PROGRAM Rotina019_Manual
VAR
	status: INT;
	
	posicaoAtual: STRING;
	envialog: STRING;
	
	fbTimeVentila: ton;
	fbTimeAqueci: ton;
	
	totalManual: STRING(255);
	tempo: STRING(255);
END_VAR

fbTimeVentila();
fbTimeAqueci();

CASE status OF

0:
IF gvl_p.arrStatusEstufas[0].startManual AND STRING_TO_DT(gvl.progInicio[0]) <= systemtime_to_dt(gvl.fbGetLocalSystemTime.systemTime)  THEN
	status:= 5;
	
	gvl.bstartchart019:= TRUE;
	gvl_p.zona1setpt_019:= gvl_p.arr_CustomTime[0,1];
	gvl_p.zona2setpt_019:= gvl_p.arr_CustomTime[0,1];
	gvl.liga_ventilacao_019:= TRUE;
	fbTimeVentila(in:= TRUE, pt:=T#1S);
	
///// GERADOR DE LOG -------------------------------------------------------------

envialog:= 'Programação Manual Iniciada ESTUFA 019';
gvl.logRegister19:= envialog;

	gvl_p.etapa_process[0] := 'Inicializando';
	
ELSE
	status:= 0;
	IF gvl_p.arrStatusEstufas[0].start THEN
		gvl_p.etapa_process[0] := gvl.progInicio[0];
	END_IF
END_IF
5:
IF fbTimeVentila.Q THEN
	status:= 10;
	gvl.liga_ventilacao_019:=FALSE;
	fbTimeVentila(in:= FALSE);
ELSE
	status:= 5;
END_IF

10:
IF gvl.ventilacao_Ligada_019 THEN
	status:= 15;
	
	gvl.liga_aquecimento_019:= TRUE;
	fbTimeAqueci(in:= TRUE, pt:= T#1S);
	
///// GERADOR DE LOG -------------------------------------------------------------

envialog:= 'Aquecendo ESTUFA 019';
gvl.logRegister19:= envialog;
	
	gvl_p.etapa_process[0] := 'Aquecendo';
	
ELSE
	status:= 10;
END_IF

15:
IF fbTimeAqueci.Q THEN
	status:= 20;
	
	gvl.liga_aquecimento_019:= FALSE;
	fbTimeAqueci(in:=false);
ELSE
	status:= 15;
END_IF

20:
IF gvl.zona1atual_019 >= gvl_p.zona1setpt_019 THEN
	status:= 30;
	
gvl.progInicio[0]:= DT_TO_STRING(gvl.somaTempo);
	
///// CALCULAR FIM DA SECAGEM E DA ARMAZENAGEM --------------------------------------------------------------------------------

totalManual:= insert('T#h',INT_TO_STRING(gvl.totalManual[0]),2);
gvl_p.arrStatusEstufas[0].inicioSecagem := STRING_TO_DT(gvl.progInicio[0]);
gvl_p.arrStatusEstufas[0].fimSecagem := STRING_TO_DT(gvl.progInicio[0]) + STRING_TO_TIME(totalManual);
gvl_P.arrStatusEstufas[0].prevFimSeca := gvl_p.arrStatusEstufas[0].fimSecagem;
//gvl_p.arrStatusEstufas[0].fimArmazenagem := gvl_p.arrStatusEstufas[0].fimSecagem + gvl_p.arrStatusEstufas[0].tempoArmazenagem ;

///// IMPRIMIR A HORA E A DATA DO INICIO DA SECAGEM ---------------------------------------------------------------------------
gvl_p.arrStatusEstufas[0].statusInicioSecagem := '';
gvl_p.arrStatusEstufas[0].statusInicioSecagem := concat(gvl_p.arrStatusEstufas[0].statusInicioSecagem,gvl.hora);
gvl_p.arrStatusEstufas[0].statusInicioSecagem := concat(gvl_p.arrStatusEstufas[0].statusInicioSecagem,':');
gvl_p.arrStatusEstufas[0].statusInicioSecagem := concat(gvl_p.arrStatusEstufas[0].statusInicioSecagem,gvl.minuto);
gvl_p.arrStatusEstufas[0].statusInicioSecagem := concat(gvl_p.arrStatusEstufas[0].statusInicioSecagem,' ');
gvl_p.arrStatusEstufas[0].statusInicioSecagem := concat(gvl_p.arrStatusEstufas[0].statusInicioSecagem,gvl.dia);
gvl_p.arrStatusEstufas[0].statusInicioSecagem := concat(gvl_p.arrStatusEstufas[0].statusInicioSecagem,'/');
gvl_p.arrStatusEstufas[0].statusInicioSecagem := concat(gvl_p.arrStatusEstufas[0].statusInicioSecagem,gvl.mes);
gvl_p.arrStatusEstufas[0].statusInicioSecagem := concat(gvl_p.arrStatusEstufas[0].statusInicioSecagem,'/');
gvl_p.arrStatusEstufas[0].statusInicioSecagem := concat(gvl_p.arrStatusEstufas[0].statusInicioSecagem,gvl.ano);

//--------------------REATOR------------------------------------

IF gravarConfigPosicao_Reator.bGravarConfigPosicao_Reator THEN
	gvl_p.arrStatusEstufas[0].inicioReator := '';
	gvl_p.arrStatusEstufas[0].inicioReator := concat(gvl_p.arrStatusEstufas[0].inicioReator,gvl.hora);
	gvl_p.arrStatusEstufas[0].inicioReator := concat(gvl_p.arrStatusEstufas[0].inicioReator,':');
	gvl_p.arrStatusEstufas[0].inicioReator := concat(gvl_p.arrStatusEstufas[0].inicioReator,gvl.minuto);
	gvl_p.arrStatusEstufas[0].inicioReator := concat(gvl_p.arrStatusEstufas[0].inicioReator,' ');
	gvl_p.arrStatusEstufas[0].inicioReator := concat(gvl_p.arrStatusEstufas[0].inicioReator,gvl.dia);
	gvl_p.arrStatusEstufas[0].inicioReator := concat(gvl_p.arrStatusEstufas[0].inicioReator,'/');
	gvl_p.arrStatusEstufas[0].inicioReator := concat(gvl_p.arrStatusEstufas[0].inicioReator,gvl.mes);
	gvl_p.arrStatusEstufas[0].inicioReator := concat(gvl_p.arrStatusEstufas[0].inicioReator,'/');
	gvl_P.arrStatusEstufas[0].inicioReator := concat(gvl_p.arrStatusEstufas[0].inicioReator,gvl.ano);
END_IF

///// DECOMPOR A VARIAVEL FIM DA SECAGEM -----------------------------------------------------------------------------------------------
gvl_p.arrStatusEstufas[0].diaSec := MID(STR:= DT_TO_STRING(gvl_p.arrStatusEstufas[0].fimSecagem) , LEN:= 2, POS:=12);
gvl_p.arrStatusEstufas[0].mesSec := MID(STR:= DT_TO_STRING(gvl_p.arrStatusEstufas[0].fimSecagem), LEN:= 2, POS:=9);
gvl_p.arrStatusEstufas[0].anoSec := MID(STR:= DT_TO_STRING(gvl_p.arrStatusEstufas[0].fimSecagem), LEN:= 2, POS:=6);
gvl_p.arrStatusEstufas[0].horaSec := MID(STR:= DT_TO_STRING(gvl_p.arrStatusEstufas[0].fimSecagem), LEN:= 2, POS:=15);
gvl_p.arrStatusEstufas[0].minutoSec := MID(STR:= DT_TO_STRING(gvl_p.arrStatusEstufas[0].fimSecagem), LEN:= 2, POS:=18);

///// IMPRIMIR A HORA E A DATA DO FIM DA SECAGEM --------------------------------------------------------------------------------------------------------
gvl_p.arrStatusEstufas[0].statusFimSecagem := '';
gvl_p.arrStatusEstufas[0].statusFimSecagem := concat(gvl_p.arrStatusEstufas[0].statusFimSecagem,gvl_p.arrStatusEstufas[0].horaSec);
gvl_p.arrStatusEstufas[0].statusFimSecagem := concat(gvl_p.arrStatusEstufas[0].statusFimSecagem,':');
gvl_p.arrStatusEstufas[0].statusFimSecagem := concat(gvl_p.arrStatusEstufas[0].statusFimSecagem,gvl_p.arrStatusEstufas[0].minutoSec);
gvl_p.arrStatusEstufas[0].statusFimSecagem := concat(gvl_p.arrStatusEstufas[0].statusFimSecagem,' ');
gvl_p.arrStatusEstufas[0].statusFimSecagem := concat(gvl_p.arrStatusEstufas[0].statusFimSecagem,gvl_p.arrStatusEstufas[0].diaSec);
gvl_p.arrStatusEstufas[0].statusFimSecagem := concat(gvl_p.arrStatusEstufas[0].statusFimSecagem,'/');
gvl_p.arrStatusEstufas[0].statusFimSecagem := concat(gvl_p.arrStatusEstufas[0].statusFimSecagem,gvl_p.arrStatusEstufas[0].mesSec);
gvl_p.arrStatusEstufas[0].statusFimSecagem := concat(gvl_p.arrStatusEstufas[0].statusFimSecagem,'/');
gvl_p.arrStatusEstufas[0].statusFimSecagem := concat(gvl_p.arrStatusEstufas[0].statusFimSecagem,gvl_p.arrStatusEstufas[0].anoSec);


///// GERADOR DE LOG -------------------------------------------------------------
envialog:= 'Inicio T1 ESTUFA 019';
gvl.logRegister19:= envialog;

gvl_p.etapa_process[0]:= 'T1';

ELSE
	IF gvl_p.arr_CustomTime[1,1] = 0 THEN
		status:= 45;
	END_IF
	status:= 20;
END_IF

30:
tempo:= insert('T#h',INT_TO_STRING(gvl_p.arr_CustomTime[1,1]),2);
IF STRING_TO_DT(gvl.progInicio[0]) + STRING_TO_TIME(tempo) = systemtime_to_dt(gvl.fbGetLocalSystemTime.systemTime) THEN
	status:= 31;
	
	gvl_p.zona1setpt_019:= gvl_p.arr_CustomTime[0,2];
	gvl_p.zona2setpt_019:= gvl_p.arr_CustomTime[0,2];
	gvl.progInicio[0]:= DT_TO_STRING(STRING_TO_DT(gvl.progInicio[0]) + STRING_TO_TIME(tempo));
	
///// GERADOR DE LOG -------------------------------------------------------------
envialog:= 'Inicio T2 ESTUFA 019';
gvl.logRegister19:= envialog;

gvl_p.etapa_process[0]:= 'T2';
	
ELSE
	status:= 30;
END_IF

31:
tempo:= insert('T#h',INT_TO_STRING(gvl_p.arr_CustomTime[1,2]),2);
IF STRING_TO_DT(gvl.progInicio[0]) + STRING_TO_TIME(tempo) = systemtime_to_dt(gvl.fbGetLocalSystemTime.systemTime) THEN
	status:= 32;
	
	gvl_p.zona1setpt_019:= gvl_p.arr_CustomTime[0,3];
	gvl_p.zona2setpt_019:= gvl_p.arr_CustomTime[0,3];
	gvl.progInicio[0]:= DT_TO_STRING(STRING_TO_DT(gvl.progInicio[0]) + STRING_TO_TIME(tempo));
	
///// GERADOR DE LOG -------------------------------------------------------------
envialog:= 'Inicio T3 ESTUFA 019';
gvl.logRegister19:= envialog;

gvl_p.etapa_process[0]:= 'T3';
	
ELSE
	IF gvl_p.arr_CustomTime[1,2] = 0 THEN
		status:= 45;
	END_IF
	status:= 31;
END_IF

32:
tempo:= insert('T#h',INT_TO_STRING(gvl_p.arr_CustomTime[1,3]),2);
IF STRING_TO_DT(gvl.progInicio[0]) + STRING_TO_TIME(tempo) = systemtime_to_dt(gvl.fbGetLocalSystemTime.systemTime) THEN
	status:= 33;
	
	gvl_p.zona1setpt_019:= gvl_p.arr_CustomTime[0,4];
	gvl_p.zona2setpt_019:= gvl_p.arr_CustomTime[0,4];
	gvl.progInicio[0]:= DT_TO_STRING(STRING_TO_DT(gvl.progInicio[0]) + STRING_TO_TIME(tempo));
	
///// GERADOR DE LOG -------------------------------------------------------------
envialog:= 'Inicio T4 ESTUFA 019';
gvl.logRegister19:= envialog;

gvl_p.etapa_process[0]:= 'T4';
	
ELSE
	IF gvl_p.arr_CustomTime[1,3] = 0 THEN
		status:= 45;
	END_IF
	status:= 32;
END_IF

33:
tempo:= insert('T#h',INT_TO_STRING(gvl_p.arr_CustomTime[1,4]),2);
IF STRING_TO_DT(gvl.progInicio[0]) + STRING_TO_TIME(tempo) = systemtime_to_dt(gvl.fbGetLocalSystemTime.systemTime) THEN
	status:= 34;
	
	gvl_p.zona1setpt_019:= gvl_p.arr_CustomTime[0,5];
	gvl_p.zona2setpt_019:= gvl_p.arr_CustomTime[0,5];
	gvl.progInicio[0]:= DT_TO_STRING(STRING_TO_DT(gvl.progInicio[0]) + STRING_TO_TIME(tempo));
	
///// GERADOR DE LOG -------------------------------------------------------------
envialog:= 'Inicio T5 ESTUFA 019';
gvl.logRegister19:= envialog;

gvl_p.etapa_process[0]:= 'T5';
	
ELSE
	IF gvl_p.arr_CustomTime[1,4] = 0 THEN
		status:= 45;
	END_IF
	status:= 33;
END_IF

34:
tempo:= insert('T#h',INT_TO_STRING(gvl_p.arr_CustomTime[1,5]),2);
IF STRING_TO_DT(gvl.progInicio[0]) + STRING_TO_TIME(tempo) = systemtime_to_dt(gvl.fbGetLocalSystemTime.systemTime) THEN
	status:= 35;
	
	gvl_p.zona1setpt_019:= gvl_p.arr_CustomTime[0,6];
	gvl_p.zona2setpt_019:= gvl_p.arr_CustomTime[0,6];
	gvl.progInicio[0]:= DT_TO_STRING(STRING_TO_DT(gvl.progInicio[0]) + STRING_TO_TIME(tempo));
	
///// GERADOR DE LOG -------------------------------------------------------------
envialog:= 'Inicio T6 ESTUFA 019';
gvl.logRegister19:= envialog;

gvl_p.etapa_process[0]:= 'T6';
	
ELSE
	IF gvl_p.arr_CustomTime[1,5] = 0 THEN
		status:= 45;
	END_IF
	status:= 34;
END_IF

35:
tempo:= insert('T#h',INT_TO_STRING(gvl_p.arr_CustomTime[1,6]),2);
IF STRING_TO_DT(gvl.progInicio[0]) + STRING_TO_TIME(tempo) = systemtime_to_dt(gvl.fbGetLocalSystemTime.systemTime) THEN
	status:= 36;
	
	gvl_p.zona1setpt_019:= gvl_p.arr_CustomTime[0,7];
	gvl_p.zona2setpt_019:= gvl_p.arr_CustomTime[0,7];
	gvl.progInicio[0]:= DT_TO_STRING(STRING_TO_DT(gvl.progInicio[0]) + STRING_TO_TIME(tempo));
	
///// GERADOR DE LOG -------------------------------------------------------------
envialog:= 'Inicio T7 ESTUFA 019';
gvl.logRegister19:= envialog;

gvl_p.etapa_process[0]:= 'T7';
	
ELSE
	IF gvl_p.arr_CustomTime[1,6] = 0 THEN
		status:= 45;
	END_IF
	status:= 35;
END_IF

36:
tempo:= insert('T#h',INT_TO_STRING(gvl_p.arr_CustomTime[1,7]),2);
IF STRING_TO_DT(gvl.progInicio[0]) + STRING_TO_TIME(tempo) = systemtime_to_dt(gvl.fbGetLocalSystemTime.systemTime) THEN
	status:= 37;
	
	gvl_p.zona1setpt_019:= gvl_p.arr_CustomTime[0,8];
	gvl_p.zona2setpt_019:= gvl_p.arr_CustomTime[0,8];
	gvl.progInicio[0]:= DT_TO_STRING(STRING_TO_DT(gvl.progInicio[0]) + STRING_TO_TIME(tempo));
	
///// GERADOR DE LOG -------------------------------------------------------------
envialog:= 'Inicio T8 ESTUFA 019';
gvl.logRegister19:= envialog;

gvl_p.etapa_process[0]:= 'T8';
	
ELSE
	IF gvl_p.arr_CustomTime[1,7] = 0 THEN
		status:= 45;
	END_IF
	status:= 36;
END_IF

37:
tempo:= insert('T#h',INT_TO_STRING(gvl_p.arr_CustomTime[1,8]),2);
IF STRING_TO_DT(gvl.progInicio[0]) + STRING_TO_TIME(tempo) = systemtime_to_dt(gvl.fbGetLocalSystemTime.systemTime) THEN
	status:= 38;
	
	gvl_p.zona1setpt_019:= gvl_p.arr_CustomTime[0,9];
	gvl_p.zona2setpt_019:= gvl_p.arr_CustomTime[0,9];
	gvl.progInicio[0]:= DT_TO_STRING(STRING_TO_DT(gvl.progInicio[0]) + STRING_TO_TIME(tempo));
	
///// GERADOR DE LOG -------------------------------------------------------------
envialog:= 'Inicio T9 ESTUFA 019';
gvl.logRegister19:= envialog;

gvl_p.etapa_process[0]:= 'T9';
	
ELSE
	IF gvl_p.arr_CustomTime[1,8] = 0 THEN
		status:= 45;
	END_IF
	status:= 37;
END_IF

38:
tempo:= insert('T#h',INT_TO_STRING(gvl_p.arr_CustomTime[1,9]),2);
IF STRING_TO_DT(gvl.progInicio[0]) + STRING_TO_TIME(tempo) = systemtime_to_dt(gvl.fbGetLocalSystemTime.systemTime) THEN
	status:= 40;
	
	gvl_p.zona1setpt_019:= gvl_p.arr_CustomTime[0,10];
	gvl_p.zona2setpt_019:= gvl_p.arr_CustomTime[0,10];
	gvl.progInicio[0]:= DT_TO_STRING(STRING_TO_DT(gvl.progInicio[0]) + STRING_TO_TIME(tempo));
	
///// GERADOR DE LOG -------------------------------------------------------------
envialog:= 'Inicio T10 ESTUFA 019';
gvl.logRegister19:= envialog;

gvl_p.etapa_process[0]:= 'T10';
	
ELSE
	IF gvl_p.arr_CustomTime[1,9] = 0 THEN
		status:= 45;
	END_IF
	status:= 38;
END_IF

40:
tempo:= insert('T#h',INT_TO_STRING(gvl_p.arr_CustomTime[1,10]),2);
IF STRING_TO_DT(gvl.progInicio[0]) + STRING_TO_TIME(tempo) = systemtime_to_dt(gvl.fbGetLocalSystemTime.systemTime) THEN
	status:= 50;
	
	gvl_p.arrStatusEstufas[0].startManual:= FALSE;
	gvl.bstartchart019:= FALSE;
	gvl.desl_aquecimento_019:= TRUE;
	fbTimeAqueci(in:=TRUE, pt:=T#1S);
	
	gvl_p.etapa_process[0] := '';
	
	gvl_p.arrStatusEstufas[0].statusInicioSecagem := '';
	gvl_p.arrStatusEstufas[0].inicioReator := '';
	gvl_p.arrStatusEstufas[0].statusFimSecagem := '';
	gvl_p.arrStatusEstufas[0].statusFimArmazenagem := '';
	gvl_p.arrStatusEstufas[0].fimSecagem:= DT#1970-1-1-0:0:0;
	gvl.endArm19:= T#0S;
	gvl.endSeca19:= T#0S;
	
///// GERADOR DE LOG -------------------------------------------------------------
envialog:= 'Programação Finalizada ESTUFA 019';
gvl.logRegister19:= envialog;

gvl_p.etapa_process[0]:= '';

ELSE
	IF gvl_p.arr_CustomTime[1,10] = 0 THEN
		status:= 45;
	END_IF
	status:= 40;
END_IF

45:
IF gvl_p.arrStatusEstufas[0].startManual THEN
status:= 50;
	
	gvl_p.arrStatusEstufas[0].startManual:= FALSE;
	gvl.bstartchart019:= FALSE;
	gvl.desl_aquecimento_019:= TRUE;
	fbTimeAqueci(in:=TRUE, pt:=T#1S);
	
	gvl_p.etapa_process[0] := '';
	
	gvl_p.arrStatusEstufas[0].statusInicioSecagem := '';
	gvl_p.arrStatusEstufas[0].inicioReator := '';
	gvl_p.arrStatusEstufas[0].statusFimSecagem := '';
	gvl_p.arrStatusEstufas[0].statusFimArmazenagem := '';
	gvl_p.arrStatusEstufas[0].fimSecagem:= DT#1970-1-1-0:0:0;
	gvl.endArm19:= T#0S;
	gvl.endSeca19:= T#0S;
	
///// GERADOR DE LOG -------------------------------------------------------------
envialog:= 'Programação Finalizada ESTUFA 019';
gvl.logRegister19:= envialog;

gvl_p.etapa_process[0]:= '';

ELSE
	status:= 45;
END_IF

50:
IF fbTimeAqueci.Q THEN
	status:= 0;
	
	gvl.desl_aquecimento_019:= FALSE;
	fbTimeAqueci(in:= FALSE);
	
ELSE
	status:= 50;
END_IF
END_CASE

END_PROGRAM

(* stored: Version 1.1.0.1, ProductVersion 3.1.4024.12
   POU Rotina019_Manual: Id {d4d8b9c9-c72d-4c7b-9bcd-a545026575a6}, SpecialFunc None *)
